FUNCTION_BLOCK SYMLINKMULTIVARDST_277E97BEC1451D2C (* Multiple variables single value symbolic link destination FB *)
  (* Standard: 61499-2 *)
  (* Version 1.0, 2008-10-02, milos, nxtControl GmbH, template *)
  PACKAGE UAO.Hackathon;
  (* Compiler Cpp *)
  {SET_ATTRIBUTE(Runtime.FBType.ImplementingType, Runtime.System#DYNGEN_SYMLINKMVAR)}
  {SET_ATTRIBUTE(Configuration.GenericFBType.InterfaceParams, Runtime.System#I:=2;VALUE${I$}:BOOL,BOOL)}
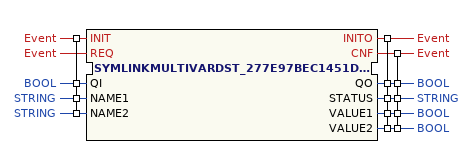
  EVENT_INPUT
    INIT WITH QI, NAME1, NAME2; (* Initializes the symbolic link data destination FB with N (1 <= N <= 16) variables *)
    REQ; (* Explicit data read request *)
  END_EVENT
  EVENT_OUTPUT
    INITO WITH QO, STATUS, VALUE1, VALUE2; (* Initialization confirm *)
    CNF WITH QO, STATUS, VALUE1, VALUE2; (* Confirmation of an explicit or implicit data read request *)
  END_EVENT
  VAR_INPUT
    QI : BOOL; (* INIT event input qualifier *)
    NAME1 : STRING := '$${PATH}'; (* Names a symbolic link variable *)
    NAME2 : STRING := '$${PATH}'; (* Names a symbolic link variable *)
  END_VAR
  VAR_OUTPUT
    QO : BOOL; (* Output event qualifier *)
    STATUS : STRING; (* FB status indicator *)
    VALUE1 : BOOL; (* Current value(i) in the named variable array element *)
    VALUE2 : BOOL; (* Current value(i) in the named variable array element *)
  END_VAR
  EC_STATES
    START;
  END_STATES
END_FUNCTION_BLOCK
